Yaskawa INFORM job: R2_W13,15(0,0)_MP_OK.JBI

/JOB
//NAME R2_W13,15(0,0)_MP_OK
///FOLDERNAME MP_TEST
//POS
///NPOS 96,96,0,5,0,0
///TOOL 0
///POSTYPE PULSE
///PULSE
C00000=160074,80797,26825,14512,73882,-11454
C00001=160843,86662,35984,14314,71214,-11522
C00002=161140,89195,39907,14253,70085,-11558
C00003=161775,90672,41778,13960,69602,-11398
C00004=161140,89195,39907,14253,70085,-11558
C00005=161063,90646,42469,14364,69291,-11681
C00006=161063,90039,43321,14440,68480,-11781
C00007=161063,90646,42469,14364,69291,-11681
C00008=160899,91716,44118,14490,68868,-11791
C00009=160588,94104,47162,14712,68294,-11972
C00010=160899,91716,44118,14490,68868,-11791
C00011=160602,89056,40019,14540,70038,-11748
C00012=159834,82934,30508,14714,72789,-11666
C00013=159775,78785,28717,31049,45785,-17949
C00014=160744,86276,37714,31059,43998,-18135
C00015=161118,89436,41574,31127,43221,-18241
C00016=161766,90979,43527,30761,42643,-18122
C00017=161118,89436,41574,31127,43221,-18241
C00018=160989,91460,44001,31494,42875,-18446
C00019=160696,93702,46857,32104,42461,-18773
C00020=160989,91460,44001,31494,42875,-18446
C00021=160955,90463,41510,30968,43766,-18115
C00022=160955,91376,40496,30399,44712,-17757
C00023=160955,90463,41510,30968,43766,-18115
C00024=160580,87312,37646,30905,44550,-18008
C00025=159608,79843,28641,30904,46351,-17821
C00026=169578,72061,52050,33550,65373,-36771
C00027=159639,102066,52849,36627,118532,-43382
C00028=161230,98010,49947,36645,117651,-43000
C00029=161874,96468,48906,36639,117269,-42855
C00030=162414,97439,51471,36313,116175,-43029
C00031=161874,96468,48906,36639,117269,-42855
C00032=161681,87636,37192,37728,115333,-39463
C00033=162202,89199,38314,37765,115213,-39280
C00034=161681,87636,37192,37728,115333,-39463
C00035=159221,89245,43122,43634,115424,-41269
C00036=159607,86334,39462,43925,115798,-40898
C00037=159221,89245,43122,43634,115424,-41269
C00038=158510,90592,44026,43670,115855,-41410
C00039=156755,94145,46551,43727,116872,-41780
C00040=156215,89463,47666,89737,91612,-44965
C00041=160258,86848,41994,88867,88907,-43909
C00042=161076,86470,41042,88663,88366,-43712
C00043=161752,88067,43044,88493,87876,-43890
C00044=161076,86470,41042,88663,88366,-43712
C00045=160594,87728,35116,82489,91621,-42752
C00046=160965,85254,32003,82415,91483,-42439
C00047=160594,87728,35116,82489,91621,-42752
C00048=161203,99397,53897,87809,93262,-46482
C00049=161203,99945,53017,87887,93322,-46099
C00050=161203,99397,53897,87809,93262,-46482
C00051=160420,100287,55440,87942,93770,-46729
C00052=156570,105790,64558,88393,96280,-48111
C00053=167330,87655,71107,35269,63189,-38515
C00054=174783,98077,26040,17019,52914,20234
C00055=174608,105356,36185,17755,50551,19749
C00056=174540,108469,40544,18090,49531,19530
C00057=174948,106579,37990,17568,50029,19783
C00058=174535,106021,37238,17896,50273,19669
C00059=174545,95141,46292,21634,39727,17290
C00060=174613,91639,41667,21115,40689,17584
C00061=174788,83471,31002,20015,42870,18217
C00062=174723,64811,15244,20023,42994,18215
C00063=174630,72581,24118,20397,41940,17819
C00064=165301,85991,63683,95469,38910,-6878
C00065=174940,70430,32149,23153,35919,16371
C00066=174503,69857,31471,23577,36151,16189
C00067=165282,98803,97625,112321,41838,-16779
C00068=174585,69363,53194,35008,24097,10312
C00069=174770,59960,41929,32247,25789,11666
C00070=174830,84723,25751,25992,31293,14140
C00071=159839,114570,69332,85586,51587,-5334
C00072=162529,132656,93679,89709,49247,-8617
C00073=174998,94453,36907,27180,29568,13493
C00074=174582,93879,36167,27626,29834,13336
C00075=152510,99797,82431,97838,56868,-14183
C00076=174570,93971,42649,20916,41255,17710
C00077=174743,85777,31872,19826,43493,18343
C00078=148864,54141,8521,56122,89229,-20941
C00079=158634,110022,45141,82267,113564,-52206
C00080=160363,104911,38709,82349,112706,-51438
C00081=159650,90621,41933,99594,103334,-56610
C00082=160497,97456,39712,80225,111807,-53659
C00083=160755,98528,41110,80015,111579,-53795
C00084=159772,85616,58768,86011,105100,-68077
C00085=160364,89778,52514,75238,109023,-59438
C00086=158635,95667,59625,74863,109814,-60259
C00087=158650,100444,49060,78741,112115,-55889
C00088=158097,97754,61839,100897,106809,-53242
C00089=159710,92289,53440,101347,105313,-52189
C00090=159988,90634,42470,94412,106524,-46277
C00091=159803,91670,52086,101491,105167,-51947
C00092=160062,92903,53649,101325,105039,-52119
C00093=159968,90319,74690,87370,106137,-56061
C00094=152319,115320,91112,71043,111185,-65415
C00095=114526,45363,13216,71043,111185,-65415
BC00000=326241,165493,546115
BC00001=326241,165493,546115
BC00002=326241,165493,546115
BC00003=326241,165493,546115
BC00004=326241,165493,546115
BC00005=326241,165493,546115
BC00006=326241,165493,546115
BC00007=326241,165493,546115
BC00008=326241,165493,546115
BC00009=326241,165493,546115
BC00010=326241,165493,546115
BC00011=326241,165493,546115
BC00012=326241,165493,546115
BC00013=350396,178832,794962
BC00014=350396,178832,794962
BC00015=350396,178832,794962
BC00016=350396,178832,794962
BC00017=350396,178832,794962
BC00018=350396,178832,794962
BC00019=350396,178832,794962
BC00020=350396,178832,794962
BC00021=350396,178832,794962
BC00022=350396,178832,794962
BC00023=350396,178832,794962
BC00024=350396,178832,794962
BC00025=350396,178832,794962
BC00026=398174,143543,1073520
BC00027=311318,165001,575189
BC00028=311318,165001,575189
BC00029=311318,165001,575189
BC00030=311318,165001,575189
BC00031=311318,165001,575189
BC00032=311318,165001,575189
BC00033=311318,165001,575189
BC00034=311318,165001,575189
BC00035=311318,165001,575189
BC00036=311318,165001,575189
BC00037=311318,165001,575189
BC00038=311318,165001,575189
BC00039=311318,165001,575189
BC00040=359964,160012,726192
BC00041=359964,160012,726192
BC00042=359964,160012,726192
BC00043=359964,160012,726192
BC00044=359964,160012,726192
BC00045=359964,160012,726192
BC00046=359964,160012,726192
BC00047=359964,160012,726192
BC00048=359964,160012,726192
BC00049=359964,160012,726192
BC00050=359964,160012,726192
BC00051=359964,160012,726192
BC00052=359964,160012,726192
BC00053=398174,157039,1073520
BC00054=388879,154573,506066
BC00055=388879,154573,506066
BC00056=388879,154573,506066
BC00057=388879,154573,506066
BC00058=388879,154573,506066
BC00059=388879,154573,506066
BC00060=388879,154573,506066
BC00061=388879,154573,506066
BC00062=378351,142558,619314
BC00063=378351,142557,619315
BC00064=378351,142557,619315
BC00065=378351,142557,619315
BC00066=378351,142557,619315
BC00067=378351,142557,520970
BC00068=378351,142557,619315
BC00069=378351,142557,619315
BC00070=389593,155475,630236
BC00071=389593,155475,630236
BC00072=389593,155475,630236
BC00073=389593,155475,630236
BC00074=389593,155475,630236
BC00075=345034,155475,630236
BC00076=389593,155475,630236
BC00077=389593,155475,630236
BC00078=354170,143700,736269
BC00079=330953,141079,472769
BC00080=330953,141079,472769
BC00081=330953,141079,472769
BC00082=330953,141079,472769
BC00083=330953,141079,472769
BC00084=330953,141080,472766
BC00085=330953,141079,472769
BC00086=330953,141079,472769
BC00087=330953,141079,472769
BC00088=331565,139590,717176
BC00089=331565,139590,717176
BC00090=331565,139590,717176
BC00091=331565,139590,717176
BC00092=331565,139590,717176
BC00093=331565,139590,717176
BC00094=331565,139590,717176
BC00095=334048,204953,873486
///POSTYPE BASE
///RECTAN
///RCONF 0,0,0,0,0,0,0,0,0,0,0,0,0,0,0,0,0,0,0,0,0,0,0,0
P00006=0.222,-3.123,-1.508,0.0000,0.0000,0.0000
P00021=-0.225,-6.128,-0.405,0.0000,0.0000,0.0000
P00022=0.222,-3.123,-1.508,0.0000,0.0000,0.0000
P00023=0.143,-0.036,0.682,0.0000,0.0000,0.0000
P00024=0.145,-0.552,1.326,0.0000,0.0000,0.0000
//INST
///DATE 2023/11/16 13:11
///ATTR SC,RW
///GROUP1 RB1,BS1
NOP
'r2_W13,15(0,0)
'
'Path S869
SFTOF
MOVJ C00000 BC00000 VJ=20.00
MOVL C00001 BC00001 V=100.0
MOVL C00002 BC00002 V=60.0
REFP 3 C00003 BC00003
CALL JOB:SEARCH-R1
SET P021 P006
SFTON P021
MOVL C00004 BC00004 V=60.0
MOVL C00005 BC00005 V=60.0
REFP 3 C00006 BC00006
CALL JOB:SEARCH-R1
SET P021 P006
SFTON P021
MOVL C00007 BC00007 V=60.0
MOVL C00008 BC00008 V=60.0
REFP 3 C00009 BC00009
CALL JOB:SEARCH-R1
SET P021 P006
SFTON P021
MOVL C00010 BC00010 V=60.0
MOVL C00011 BC00011 V=100.0
MOVL C00012 BC00012 V=100.0
'Path S870 (for W413)
SFTOF
MOVL C00013 BC00013 V=100.0
MOVL C00014 BC00014 V=100.0
MOVL C00015 BC00015 V=60.0
REFP 3 C00016 BC00016
CALL JOB:SEARCH-R1
SET P022 P006
SFTON P022
MOVL C00017 BC00017 V=60.0
MOVL C00018 BC00018 V=60.0
REFP 3 C00019 BC00019
CALL JOB:SEARCH-R1
SET P022 P006
SFTON P022
MOVL C00020 BC00020 V=60.0
MOVL C00021 BC00021 V=60.0
REFP 3 C00022 BC00022
CALL JOB:SEARCH-R1
SET P022 P006
SFTON P022
MOVL C00023 BC00023 V=60.0
MOVL C00024 BC00024 V=100.0
MOVL C00025 BC00025 V=100.0
MOVJ C00026 BC00026 VJ=20.00
'Path S871 (for W414)
'ZLA KOLEJNOSC
SFTOF
MOVL C00027 BC00027 V=100.0
MOVL C00028 BC00028 V=100.0
MOVL C00029 BC00029 V=60.0
REFP 3 C00030 BC00030
CALL JOB:SEARCH-R1
SET P023 P006
SFTON P023
MOVL C00031 BC00031 V=60.0
MOVL C00032 BC00032 V=60.0
REFP 3 C00033 BC00033
CALL JOB:SEARCH-R1
SET P023 P006
SFTON P023
MOVL C00034 BC00034 V=60.0
MOVL C00035 BC00035 V=60.0
REFP 3 C00036 BC00036
CALL JOB:SEARCH-R1
SET P023 P006
SFTON P023
MOVL C00037 BC00037 V=60.0
MOVL C00038 BC00038 V=100.0
MOVL C00039 BC00039 V=100.0
'Path S872 (for W414)
SFTOF
MOVJ C00040 BC00040 VJ=20.00
MOVL C00041 BC00041 V=100.0
MOVL C00042 BC00042 V=60.0
REFP 3 C00043 BC00043
CALL JOB:SEARCH-R1
SET P024 P006
SFTON P024
MOVL C00044 BC00044 V=60.0
MOVL C00045 BC00045 V=60.0
REFP 3 C00046 BC00046
CALL JOB:SEARCH-R1
SET P024 P006
SFTON P024
MOVL C00047 BC00047 V=60.0
MOVL C00048 BC00048 V=60.0
REFP 3 C00049 BC00049
CALL JOB:SEARCH-R1
SET P024 P006
SFTON P024
MOVL C00050 BC00050 V=60.0
MOVL C00051 BC00051 V=100.0
MOVL C00052 BC00052 V=100.0
MOVJ C00053 BC00053 VJ=20.00
COMM 'Path W873
COMM SFTOF
COMM SFTON P022
COMM MOVJ C00054 BC00054 VJ=100.00
COMM MOVL C00055 BC00055 V=400.0
COMM MOVL C00056 BC00056 V=100.0 PL=0
COMM REFP 1 C00057 BC00057
COMM REFP 2 C00058 BC00058
COMM MACRO1 MJ#(0) ARGF0
COMM ARCON
COMM SFTON P021
COMM MOVL C00059 BC00059 V=10.0
COMM ARCOF
COMM MOVL C00060 BC00060 V=400.0
COMM MOVL C00061 BC00061 V=1000.0
COMM SFTOF
'Path W916
SFTOF
SFTON P022
MOVJ C00062 BC00062 VJ=20.00
MOVL C00063 BC00063 V=100.0
MOVL C00064 BC00064 V=100.0 PL=0
REFP 1 C00065 BC00065
REFP 2 C00066 BC00066
MACRO1 MJ#(0) ARGF9
ARCON
SFTON P021
MOVL C00067 BC00067 V=11.7
ARCOF
MOVL C00068 BC00068 V=100.0
MOVL C00069 BC00069 V=100.0
SFTOF
'Path W917
SFTOF
SFTON P022
MOVJ C00070 BC00070 VJ=20.00
MOVL C00071 BC00071 V=100.0
MOVL C00072 BC00072 V=100.0 PL=0
REFP 1 C00073 BC00073
REFP 2 C00074 BC00074
MACRO1 MJ#(0) ARGF9
ARCON
MOVL C00075 BC00075 V=11.7
ARCOF
MOVL C00076 BC00076 V=100.0
MOVL C00077 BC00077 V=100.0
SFTOF
'Path VIA920
SFTOF
MOVJ C00078 BC00078 VJ=20.00
'Path W918
SFTOF
SFTON P024
MOVJ C00079 BC00079 VJ=20.00
MOVL C00080 BC00080 V=100.0
MOVL C00081 BC00081 V=100.0 PL=0
REFP 1 C00082 BC00082
REFP 2 C00083 BC00083
MACRO1 MJ#(0) ARGF10
ARCON
SFTON P023
MOVL C00084 BC00084 V=9.2
ARCOF
MOVL C00085 BC00085 V=100.0
MOVL C00086 BC00086 V=100.0
MOVL C00087 BC00087 V=100.0
SFTOF
'Path W919
SFTOF
SFTON P024
MOVJ C00088 BC00088 VJ=20.00
MOVL C00089 BC00089 V=100.0
MOVL C00090 BC00090 V=100.0 PL=0
REFP 1 C00091 BC00091
REFP 2 C00092 BC00092
MACRO1 MJ#(0) ARGF10
ARCON
MOVL C00093 BC00093 V=9.2
SFTON P023
ARCOF
MOVL C00094 BC00094 V=100.0
MOVJ C00095 BC00095 VJ=20.00
SFTOF
END
